FUNCTION_BLOCK CylinderCtrl (* Template for a simple Basic Function Block Type *)
  (* Standard: 61499-2 *)
  (* Version 1.0, 2018-07-09, az *)
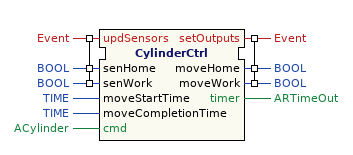
  EVENT_INPUT
    updSensors WITH senHome, senWork;
  END_EVENT
  EVENT_OUTPUT
    setOutputs WITH moveHome, moveWork;
  END_EVENT
  VAR_INPUT
    senHome : BOOL;
    senWork : BOOL;
    moveStartTime : TIME; (* timeout value till a move should start *)
    moveCompletionTime : TIME; (* timeout till a full movement completes *)
  END_VAR
  VAR_OUTPUT
    moveHome : BOOL;
    moveWork : BOOL;
  END_VAR
  SOCKETS
    cmd : ACylinder; (* Command interface for requesting cylinder actions *)
  END_SOCKETS
  PLUGS
    timer : ARTimeOut;
  END_PLUGS
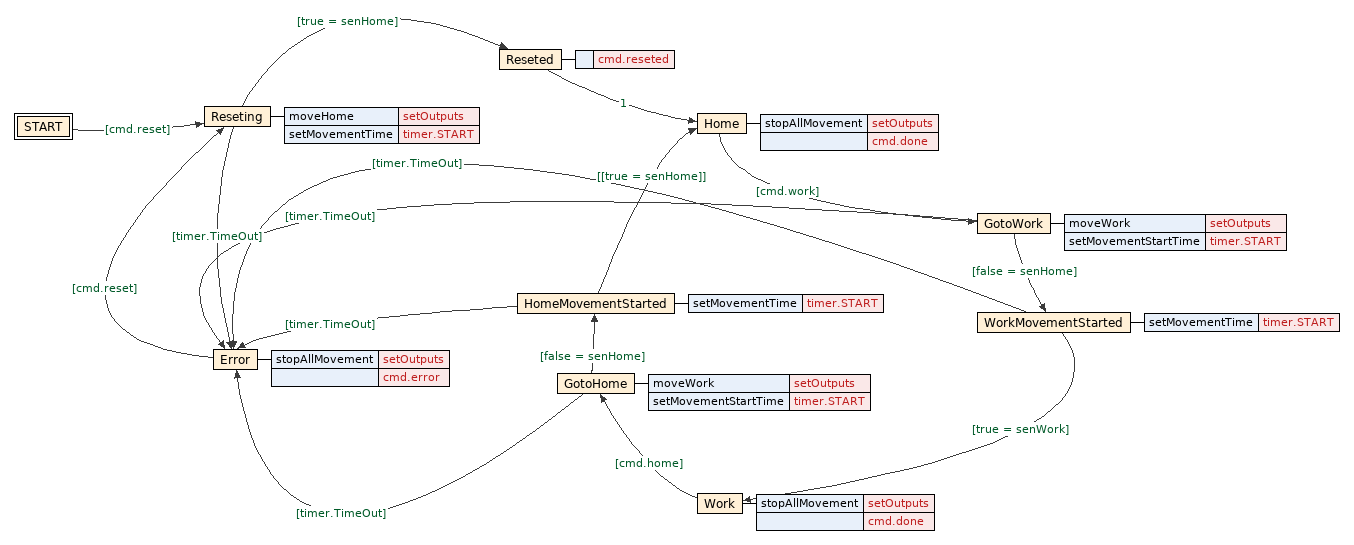
  EC_STATES
    START; (* Initial State *)
    Reseting : moveHome -> setOutputs, setMovementTime -> timer.START; (* Initialization *)
    Error : stopAllMovement -> setOutputs, -> cmd.error;
    Home : stopAllMovement -> setOutputs, -> cmd.done;
    Work : stopAllMovement -> setOutputs, -> cmd.done;
    Reseted : -> cmd.reseted;
    GotoWork : moveWork -> setOutputs, setMovementStartTime -> timer.START;
    WorkMovementStarted : setMovementTime -> timer.START;
    GotoHome : moveWork -> setOutputs, setMovementStartTime -> timer.START;
    HomeMovementStarted : setMovementTime -> timer.START;
  END_STATES
  EC_TRANSITIONS
    START TO Reseting := [cmd.reset];
    Error TO Reseting := [cmd.reset];
    Reseted TO Home := 1;
    Reseting TO Reseted := [true = senHome];
    Reseting TO Error := [timer.TimeOut];
    GotoWork TO WorkMovementStarted := [false = senHome];
    WorkMovementStarted TO Work := [true = senWork];
    Home TO GotoWork := [cmd.work];
    GotoWork TO Error := [timer.TimeOut];
    WorkMovementStarted TO Error := [timer.TimeOut];
    Work TO GotoHome := [cmd.home];
    GotoHome TO HomeMovementStarted := [false = senHome];
    HomeMovementStarted TO Home := [[true = senHome]];
    HomeMovementStarted TO Error := [timer.TimeOut];
    GotoHome TO Error := [timer.TimeOut];
  END_TRANSITIONS
  ALGORITHM moveHome IN ST: (* Initialization algorithm *)
moveHome := true;
moveWork := false;
  END_ALGORITHM
  ALGORITHM moveWork IN ST: (* Normally executed algorithm *)
moveHome := false;
moveWork := true;
  END_ALGORITHM
  ALGORITHM setMovementStartTime IN ST: (* new algorithm *)
timer.DT := moveStartTime;
  END_ALGORITHM
  ALGORITHM setMovementTime IN ST: (* new algorithm *)
timer.DT := moveCompletionTime;
  END_ALGORITHM
  ALGORITHM stopAllMovement IN ST: (* new algorithm *)
moveHome := false;
moveWork := false;
  END_ALGORITHM
END_FUNCTION_BLOCK
